# EPICS autosave request: xx_auto_dac_positions.req
$(P)$(DAC)_1.VAL
$(P)$(DAC)_2.VAL
$(P)$(DAC)_3.VAL
$(P)$(DAC)_4.VAL
$(P)$(DAC)_5.VAL
$(P)$(DAC)_6.VAL
$(P)$(DAC)_7.VAL
$(P)$(DAC)_8.VAL
